{attribute 'GeneratedUsingTerminal: EL2596-0000-0017'}
{attribute addProperty BoxType "EL2596-0000-0017"}
{attribute addProperty Description "EL2596 1-channel LED strobe control terminal 24V/3A"}
{attribute addProperty Physics "KK"}
{attribute addProperty Id "DOX_StatusAT %I*DOX_Status_F52B34D37DOX_ControlAT %Q*DOX_Control_B191BB935WcStateAT %I*WcState_9091E0EB2InfoDataAT %I*InfoData_32EB74EA10"}
{attribute addProperty CRC "234542965"}
{attribute addProperty Size "24"}
TYPE EL2596_0DFAD775 EXTENDS EtcSlaveTerminalBase_947E5A46 :
STRUCT
	{attribute addProperty Name "DOX_Status"}
	DOX_Status : DOX_Status_F52B34D3;
	{attribute addProperty Name "DOX_Control"}
	DOX_Control : DOX_Control_B191BB93;
	{attribute addProperty Name "WcState"}
	WcState : WcState_9091E0EB;
	{attribute addProperty Name "InfoData"}
	InfoData : InfoData_32EB74EA;
END_STRUCT
END_TYPE

(* stored: Version 1.2.0.0, ProductVersion 3.1.4024.11
   DUT EL2596_0DFAD775: Id {9a315e59-e7c9-40c9-a9fb-f2e4bbe62a1b} *)
